(* IEC 61131-3 sources: eCockpitGit/test_project/src/%F%00 Library/%F%Common Functions/%F%Dynamic Array/%POU%FB_DynamicArray/%PRO%getArray, 1 file *)

(* ---- %GETSET%Get.st ---- *)
VAR
END_VAR

(*%!%__DELIMITER__%!%*)
getArray		:=		S_array^;
